FUNCTION_BLOCK Encoder
VAR_INPUT
END_VAR
VAR_OUTPUT
END_VAR
VAR
	wDeviceAddress : WORD;
	iPositionActual : INT;
	iSpeedActual : INT;
END_VAR

METHOD FB_init : BOOL
VAR_INPUT
	bInitRetains : BOOL; // if TRUE, the retain variables are initialized (warm start / cold start)
	bInCopyCode : BOOL;  // if TRUE, the instance afterwards gets moved into the copy code (online change)
END_VAR
END_METHOD

PROPERTY PUBLIC positionActual : INT
GET
positionActual := iPositionActual;
END_GET
END_PROPERTY

PROPERTY PUBLIC speedActual : INT
GET
speedActual := iSpeedActual;
END_GET
END_PROPERTY

END_FUNCTION_BLOCK

(* stored: Version 1.1.0.1, ProductVersion 3.1.4024.12
   POU Encoder: Id {85234f50-7c39-4776-ac04-f3a6395be5ff}, SpecialFunc None
   Method FB_init: Id {f536c7cb-8993-48b6-a9d5-440984451fb5}
   Property positionActual: Id {24150512-b388-4902-8feb-3d2276216947}
   Get Get: Id {2a27a6fa-dd14-4fc1-90c4-376b827dd1f0}
   Property speedActual: Id {6618547a-e072-4256-b1ed-ecf77e465e0f}
   Get Get: Id {916b8fcf-b1d1-4ef1-98fc-6532e75ac4de} *)
